PROGRAM MAIN
VAR
END_VAR

// from VM

// hello on line 3 from VM

END_PROGRAM

(* stored: Version 1.1.0.1, ProductVersion 3.1.4024.11
   POU MAIN: Id {0f9c529a-d7ec-48ec-84d4-0c75a4c17f53}, SpecialFunc None *)
